// TIA Portal V17 export
// export: Created 2024-06-25T12:57:17.775261Z, ExportSetting WithDefaults, DisplayName Totally Integrated Automation Portal, DisplayVersion V17 Update 6, DisplayName TIA Portal Openness, DisplayVersion V17 Update 6, DisplayName TIA Portal Version Control Interface, DisplayVersion V17, DisplayName STEP 7 Professional, DisplayVersion V17 Update 6, DisplayName STEP 7 Safety, DisplayVersion V17 Update 6, DisplayName WinCC Advanced, DisplayVersion V17 Update 6
FUNCTION "Pulsadores" : Void   // FC2, LAD
{ S7_Optimized_Access := 'TRUE' }
VERSION : 0.1
// stored: AutoNumber true, IsIECCheckEnabled false, SetENOAutomatically false, UDAEnableTagReadback false
BEGIN

REGION Network 1: PULSADOR OFF
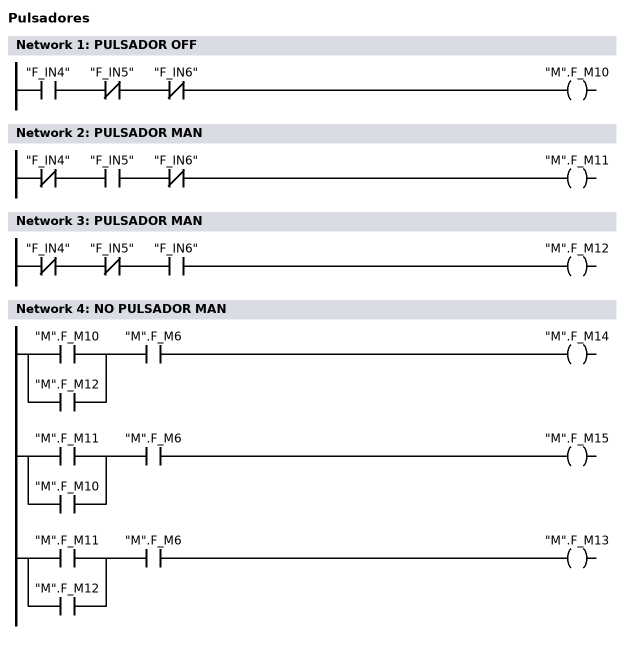
   RUNG wire#powerrail
      Contact( "F_IN4" )
      I_Contact( "F_IN5" )
      I_Contact( "F_IN6" )
      Coil( "M".F_M10 )
   END_RUNG
   // the same network as SCL:
   "M".F_M10 := "F_IN4" AND NOT "F_IN5" AND NOT "F_IN6";
END_REGION

REGION Network 2: PULSADOR MAN
   RUNG wire#powerrail
      I_Contact( "F_IN4" )
      Contact( "F_IN5" )
      I_Contact( "F_IN6" )
      Coil( "M".F_M11 )
   END_RUNG
   // the same network as SCL:
   "M".F_M11 := NOT "F_IN4" AND "F_IN5" AND NOT "F_IN6";
END_REGION

REGION Network 3: PULSADOR MAN
   RUNG wire#powerrail
      I_Contact( "F_IN4" )
      I_Contact( "F_IN5" )
      Contact( "F_IN6" )
      Coil( "M".F_M12 )
   END_RUNG
   // the same network as SCL:
   "M".F_M12 := NOT "F_IN4" AND NOT "F_IN5" AND "F_IN6";
END_REGION

REGION Network 4: NO PULSADOR MAN
   RUNG wire#powerrail
      Contact( "M".F_M10 )
      wire#w1
      Contact( "M".F_M6 )
      Coil( "M".F_M14 )
   END_RUNG
   RUNG wire#powerrail
      Contact( "M".F_M12 )
   END_RUNG wire#w1
   RUNG wire#powerrail
      Contact( "M".F_M11 )
      wire#w2
      Contact( "M".F_M6 )
      Coil( "M".F_M15 )
   END_RUNG
   RUNG wire#powerrail
      Contact( "M".F_M10 )
   END_RUNG wire#w2
   RUNG wire#powerrail
      Contact( "M".F_M11 )
      wire#w3
      Contact( "M".F_M6 )
      Coil( "M".F_M13 )
   END_RUNG
   RUNG wire#powerrail
      Contact( "M".F_M12 )
   END_RUNG wire#w3
   // the same network as SCL:
   "M".F_M14 := ("M".F_M10 OR "M".F_M12) AND "M".F_M6;
   "M".F_M15 := ("M".F_M11 OR "M".F_M10) AND "M".F_M6;
   "M".F_M13 := ("M".F_M11 OR "M".F_M12) AND "M".F_M6;
END_REGION
END_FUNCTION
